// TIA Portal V17 export
// export: Created 2023-12-22T15:03:18.9485162Z, ExportSetting WithDefaults, DisplayName Totally Integrated Automation Portal, DisplayVersion V17, DisplayName TIA Portal Openness, DisplayVersion V17, DisplayName TIA Portal Version Control Interface, DisplayVersion V17, DisplayName STEP 7 Professional, DisplayVersion V17, DisplayName STEP 7 Safety, DisplayVersion V17, DisplayName WinCC Advanced, DisplayVersion V17
DATA_BLOCK "Comm_DB"   // DB10
{ S7_Optimized_Access := 'FALSE' }
VERSION : 0.1
// stored: AutoNumber false, DBAccessibleFromOPCUA true, DBAccessibleFromWebserver true, IsOnlyStoredInLoadMemory false, IsWriteProtectedInAS false
   VAR
      SHUSKV : Array[1..11] of Struct
         Input : Struct
            DI_AllBlock : Bool;   // DI Аварийный останов
            DI_3FOk : Bool;   // DI Питание в норме
            DI_Leak_KP : Bool;   // DI Затопление камеры КП
            DI_Leak_KP_1 : Bool;   // DI Затопление камеры КП
            DI_Leak_KP_2 : Bool;   // DI Затопление камеры КП
            DI_Level_Norm : Bool;   // DI Уровень в норме
            DI_3Fok_1 : Bool;   // DI 3ф. сети Ввод 1 в норме
            DI_3Fok_2 : Bool;   // DI 3ф. сети Ввод 2 в норме
            DI_3Fok_sh : Bool;   // DI 3ф. сети Ввод Шин в норме
            DI_SHUSKV_Ok : Bool;   // DI Выключатель UC. Питание ШУСКВ в норме
            SKV_Local : Bool;   // Локальный режим скважника
            SKV_Use : Bool;   // Использование скважины
            SKV_Reset_All : Bool;   // Сброс аварий
            SKV_Pump_Ready : Bool;   // Готовность насоса
            SKV_Pump_Start : Bool;   // Запуск насоса
            SKV_Pump_Mode : Bool;   // 0 - Работа по ГЦ, 1 - Работа по расходу
            Pump_Status : Int;   // Статус насоса
            Z_1_Status : Int;   // Статус задвижки (Скважинная)
            Z_2_Status : Int;   // Статус задвижки (КП)
            Z_3_Status : Int;   // Статус задвижки (КП)
            Z_4_Status : Int;   // Статус задвижки (КП)
            Z_5_Status : Int;   // Статус задвижки (КП)
            Z_6_Status : Int;   // Статус задвижки (КП)
            Z_7_Status : Int;   // Статус задвижки (КП)
            Z_8_Status : Int;   // Статус задвижки (КП)
            Z_9_Status : Int;   // Статус задвижки (КП)
            Z_10_Status : Int;   // Статус задвижки (КП)
            Pump_OpTime_h : DInt;   // Наработка насоса
            SKV_Effect : Real;
            SKV_Distance : Real;   // Расстояние от ЩКД до скважины
            SKV_RM_SP : Real;   // Уставка для работы насоса
            SKV_Pump_SP : Real;   // Уставка производительности насоса
            AI_Cur_Pump_Result : Real;   // AI Ток двигателя насоса
            AI_LE_Result : Real;   // AI Показания уровня
            AI_PE_1_Result : Real;   // AI Показания давления 1
            AI_PE_2_Result : Real;   // AI Показания давления 2
            AI_PE_3_Result : Real;   // AI Показания давления 3
            AI_PE_4_Result : Real;   // AI Показания давления 4
            AI_TE_Result : Real;   // AI Показания температуры
            AI_Cur_Pump_Alarms : Word;   // AI Ток двигателя насоса слово аварий
            AI_LE_Alarms : Word;   // AI Слово аварий уровня
            AI_PE_1_Alarms : Word;   // AI Слово аварий давления 1
            AI_PE_2_Alarms : Word;   // AI Слово аварий давления 2
            AI_PE_3_Alarms : Word;   // AI Слово аварий давления 3
            AI_PE_4_Alarms : Word;   // AI Слово аварий давления 4
            AI_TE_Alarms : Word;   // AI Слово аварий температуры
            Pump_Alarms : Word;   // Слово аварий насоса
            Logick_Alarms : Word;   // Аварии скважины
            AI_RM_Result : Real;   // Расходомер
            SKV_Level_Norm : Real;   // Рабочая точка насоса по уровню
            SKV_LE_Skvaz : Real;
            res_1 : Word;
            res_2 : Word;
            res_3 : Word;
         END_STRUCT;
         Output : Struct
            SKV_Pump_Start : Bool;   // Запуск насоса
            SKV_Reset_All : Bool;   // Сброс аварий
            SKV_Pump_Mode : Bool;   // 0 - Работа по ГЦ, 1 - Работа по расходу
            SKV_RM_SP : Real;   // Уставка для работы насоса
            SKV_Pump_SP : Real;   // Уставка производительности насоса
            AI_LE_105_Result : Real;
            AI_LE_106_Result : Real;
            AI_LE_107_Result : Real;
            AI_LE_108_Result : Real;
            AI_TE_101_Result : Real;
            AI_TE_102_Result : Real;
            AI_TE_103_Result : Real;
            AI_TE_104_Result : Real;
            SKV_Level_Norm : Real;   // Рабочая точка насоса по уровню
            res_1 : Word;
            res_2 : Word;
            res_3 : Word;
            res_4 : Word;
            res_5 : Word;
         END_STRUCT;
      END_STRUCT;
   END_VAR
BEGIN
END_DATA_BLOCK
